FUNCTION_BLOCK AxisModTestSuite
VAR
	StubAxis : AXIS_REF;
	iStubTask : I_Task;
	TestAxisMod : MoveModTask := (AxisRef := stubaxis);
	TestObjRunner : ObjectRunner<99>;
	ObjTestSuite : TestSuite<TestSuiteParameter.MaxTestCount>(ResultFile := JUnitResultFile) := (TestSuiteName := 'Object Test Suite');
END_VAR

CheckCorrectRegistration_Test();
TaskAcceptValidCommand_Test();
TaskRejectsZeroVeloCommand_Test();

METHOD CheckCorrectRegistration_Test : BOOL
VAR_INST
	Expected : BOOL := TRUE;
	Actual	 : bool;
END_VAR
IF ObjTestSuite.Test(__POUNAME()).ExecuteTest() THEN
	TestAxisMod.RegisterWithParent(TestObjRunner);
	Actual := TestObjRunner.CyclicModuleCount = TestObjRunner.AbortableModuleCount AND
				TestObjRunner.CyclicModuleCount = TestObjRunner.TaskModuleCount;
	ObjTestSuite.Test(__POUNAME()).AssertEqual(Expected, Actual);
END_IF
END_METHOD

METHOD TaskAcceptValidCommand_Test : BOOL
VAR_INST
	Expected : BOOL := TRUE;
	Actual	 : BOOL;
END_VAR
IF ObjTestSuite.Test(__POUNAME()).ExecuteTest() THEN
	Actual := SUCCEEDED(TestAxisMod.MoveTo(100.0, 300.0));
	TestAxisMod.Abort();
	ObjTestSuite.Test(__POUNAME()).AssertEqual(Expected, Actual);
END_IF
END_METHOD

METHOD TaskRejectsZeroVeloCommand_Test : BOOL
VAR_INST
	Expected : BOOL := TRUE;
	Actual	 : BOOL;
END_VAR
IF ObjTestSuite.Test(__POUNAME()).ExecuteTest() THEN
	Actual := FAILED(TestAxisMod.MoveTo(100.0, 0.0));
	TestAxisMod.Abort();
	ObjTestSuite.Test(__POUNAME()).AssertEqual(Expected, Actual);
END_IF
END_METHOD

END_FUNCTION_BLOCK

(* stored: Version 1.1.0.1
   POU AxisModTestSuite: Id {6a9f2095-c181-4878-b784-361c97a62c94}, SpecialFunc None
   Method CheckCorrectRegistration_Test: Id {60c66d21-cbe0-4b18-b0d5-e77338525ebf}
   Method TaskAcceptValidCommand_Test: Id {b2a63fab-2531-4107-8183-36161e169aff}
   Method TaskRejectsZeroVeloCommand_Test: Id {4c4b43a6-0614-4309-af14-de1d58e6c625} *)
